PROGRAM Manipulator
VAR
	ZManipulatorMovement: RS;
	ManipulatorMovingZTrig: F_TRIG;
	CompleteSequenceOfXCounter: CTU;
	ManipulatorMovingXTrig: F_TRIG;
	XManipulatorMovement: RS;
	
	CompleteSequenceOfZCounter: CTU;
END_VAR

ManipulatorMovingZTrig(CLK:=gvl.IsManipulatorMvoingZ , Q=> );
ManipulatorMovingXTrig(CLK:=gvl.IsManipulatorMovingX , Q=> );	
CompleteSequenceOfXCounter(
	CU:=ManipulatorMovingXTrig.Q , 
	RESET:= (gvl.IsBaseClamped AND gvl.IsLidClamped) OR gvl.ResetAfterEmergency , 
	PV:=3 , 
	Q=> , 
	CV=> );
CompleteSequenceOfZCounter(
	CU:=ManipulatorMovingZTrig.Q , 
	RESET:= gvl.IsProductLeaving OR gvl.ResetAfterEmergency , 
	PV:=2 , 
	Q=> , 
	CV=> );
CASE  GVL.CurrentRobotState OF
	ManipulatorStates.WaitingToStart:
	gvl.ManipulatorXMotor:=FALSE;
	gvl.ManipulatorGrabMotor:=FALSE;
	gvl.ManipulatorZMotor:=FALSE;
	ManipulatorStates.WaitingForALid:
	
	gvl.ManipulatorGrabMotor:=FALSE;
	gvl.ManipulatorZMotor:=FALSE;
	IF gvl.IsBaseClamped AND gvl.IsLidClamped THEN
		GVL.CurrentRobotState:=ManipulatorStates.Pciking;
	END_IF
	ManipulatorStates.Pciking:
	
	IF  gvl.IsManipulatorDectectingAnObject THEN
		Gvl.ManipulatorGrabMotor:=TRUE;
	END_IF
		
	ZManipulatorMovement(SET:=(gvl.IsBaseClamped AND gvl.IsLidClamped AND NOT CompleteSequenceOfXCounter.Q ) , RESET1:=(gvl.IsManipulatorDectectingAnObject OR ManipulatorMovingZTrig.Q)   , Q1=>gvl.ManipulatorZMotor) ;
	gvl.LidClampMotor:=ZManipulatorMovement.Q1;
	IF ManipulatorMovingZTrig.Q THEN
		Gvl.LidClampMotor:=FALSE;
		GVL.CurrentRobotState:=ManipulatorStates.Placing;
	END_IF
	ManipulatorStates.Placing:
	
	XManipulatorMovement(SET:= gvl.IsBaseClamped , RESET1:=ManipulatorMovingXTrig.Q , Q1=>gvl.ManipulatorXMotor );
	ZManipulatorMovement(SET:=CompleteSequenceOfXCounter.CV=1 , RESET1:=CompleteSequenceOfZCounter.CV=2  , Q1=>gvl.ManipulatorZMotor) ;
	
	IF CompleteSequenceOfZCounter.CV=2 THEN
		gvl.CurrentBaseState:=BaseStates.Departure;
		gvl.CurrentRobotState:=ManipulatorStates.WaitingForALid;		
	END_IF
	
	ManipulatorStates.Stop:
	gvl.ManipulatorXMotor:=FALSE;
	gvl.ManipulatorGrabMotor:=FALSE;
	gvl.ManipulatorZMotor:=FALSE;
	
END_CASE

END_PROGRAM

(* stored: Version 1.1.0.1, ProductVersion 3.1.4024.9
   POU Manipulator: Id {126a1d86-8bce-428c-849c-2af7c63ae827}, SpecialFunc None *)
